// TIA Portal V20 export
TYPE "typeEm5Commands"
// stored: Access Published, Namespace Unit1
   STRUCT
      Spare { ExternalWritable := 'False'} : Bool;
   END_STRUCT;
END_TYPE
